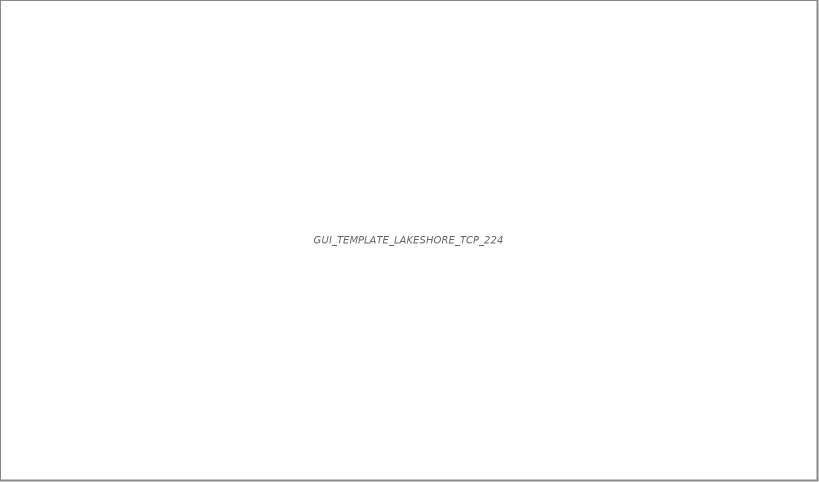
VISUALIZATION GUI_LAKESHORE_TCP_224  // 819x482
    Frame (0,0 817x480)
        shows GUI_TEMPLATE_LAKESHORE_TCP_224(m_Instance := MAIN.LS224_TCP)
END_VISUALIZATION

(* stored: Version 1.1.0.1, ProductVersion 3.1.4022.16
   Visu GUI_LAKESHORE_TCP_224: Id {2f71650d-89a0-4c1d-974b-263cb2350778} *)
